FUNCTION InstrumentReading_420mA : REAL
(*
* Takes the DAQ's curInput (unitless) and coverts to EU (mA)
* Built for use with EL3114 15 bit resolution
* Change internal variable 
* @param icurInput (INT): Raw data from ADC
* Output rcurOutput (REAL): EU real output
*)
VAR_INPUT
	icurInput : INT;
END_VAR
VAR
	rconvFactor : REAL := 16.0/(26300.0); //Will also convert int to real
END_VAR

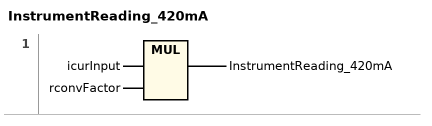
// NETWORK 1
InstrumentReading_420mA := icurInput * rconvFactor;

END_FUNCTION

(* stored: Version 1.1.0.1, ProductVersion 3.1.4024.12
   POU InstrumentReading_420mA: Id {1ac814da-fc8c-4c33-ae59-99b6aebedf22}, SpecialFunc None *)
